% RSLogix 500 project Project_8.RSS, saved by version 8.30.00.16 %
PROJECT "UNTITLED"    % processor: Bul.1763 MicroLogix 1100 Series B %

PROGRAM FILES
  LAD 2   16 rungs

DATA FILES
  O0 OUTPUT  4 elements
  I1 INPUT  6 elements
  S2 STATUS  66 elements
  B3 BINARY  1 elements
  T4 TIMER  1 elements
  C5 COUNTER  1 elements
  R6 CONTROL  1 elements
  N7 INTEGER  7 elements
  F8 FLOAT  1 elements

LADDER 2
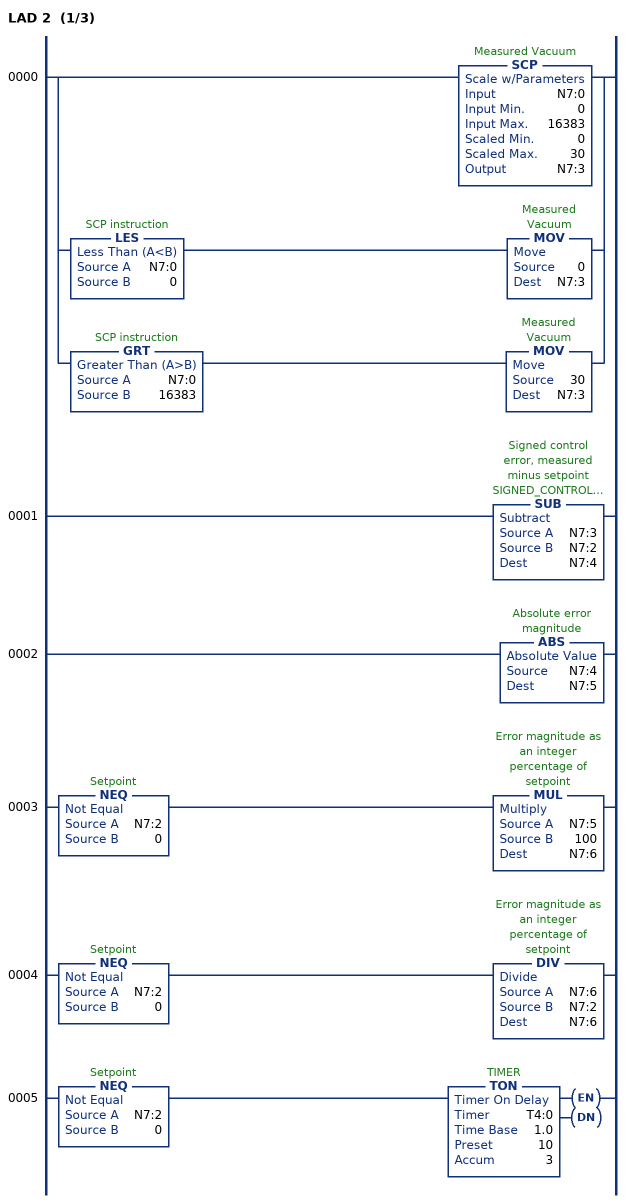
% Rung: 0 %
SOR BST SCP N7:0 0 16383 0 30 N7:3 NXB LES N7:0 0 MOV 0 N7:3 NXB GRT N7:0 16383 MOV 30 N7:3 BND EOR
%   N7:0  "SCP instruction" %
%   N7:3  "Measured Vacuum" %
% Rung: 1 %
SOR SUB N7:3 N7:2 N7:4 EOR
%   N7:3  "Measured Vacuum" %
%   N7:2  "Setpoint" %
%   N7:4  SIGNED_CONTROL_ERROR  "Signed control error, measured minus setpoint" %
% Rung: 2 %
SOR ABS N7:4 N7:5 EOR
%   N7:4  SIGNED_CONTROL_ERROR  "Signed control error, measured minus setpoint" %
%   N7:5  "Absolute error magnitude" %
% Rung: 3 %
SOR NEQ N7:2 0 MUL N7:5 100 N7:6 EOR
%   N7:2  "Setpoint" %
%   N7:5  "Absolute error magnitude" %
%   N7:6  "Error magnitude as an integer percentage of setpoint" %
% Rung: 4 %
SOR NEQ N7:2 0 DIV N7:6 N7:2 N7:6 EOR
%   N7:2  "Setpoint" %
%   N7:6  "Error magnitude as an integer percentage of setpoint" %
% Rung: 5 %
SOR NEQ N7:2 0 TON T4:0 1.0 10 3 EOR
%   N7:2  "Setpoint" %
%   T4:0  TIMER %

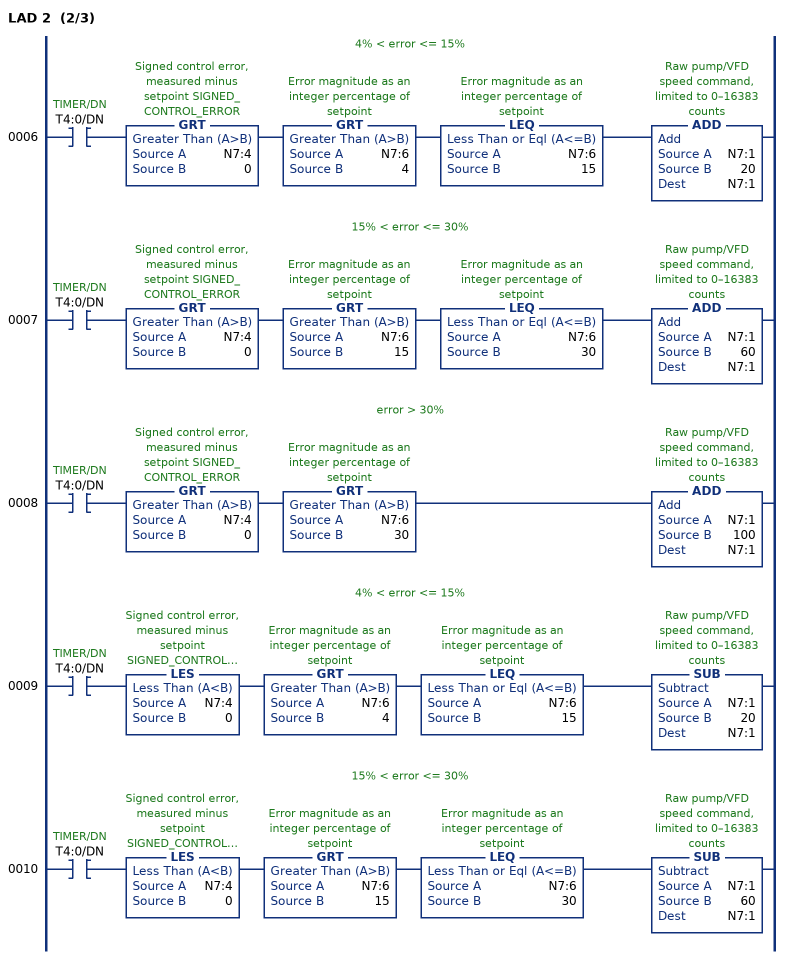
% Rung: 6 %
% 4% < error <= 15% %
SOR XIC T4:0/DN GRT N7:4 0 GRT N7:6 4 LEQ N7:6 15 ADD N7:1 20 N7:1 EOR
%   T4:0  TIMER %
%   N7:4  SIGNED_CONTROL_ERROR  "Signed control error, measured minus setpoint" %
%   N7:6  "Error magnitude as an integer percentage of setpoint" %
%   N7:1  "Raw pump/VFD speed command, limited to 0–16383 counts" %
% Rung: 7 %
% 15% < error <= 30% %
SOR XIC T4:0/DN GRT N7:4 0 GRT N7:6 15 LEQ N7:6 30 ADD N7:1 60 N7:1 EOR
%   T4:0  TIMER %
%   N7:4  SIGNED_CONTROL_ERROR  "Signed control error, measured minus setpoint" %
%   N7:6  "Error magnitude as an integer percentage of setpoint" %
%   N7:1  "Raw pump/VFD speed command, limited to 0–16383 counts" %
% Rung: 8 %
% error > 30% %
SOR XIC T4:0/DN GRT N7:4 0 GRT N7:6 30 ADD N7:1 100 N7:1 EOR
%   T4:0  TIMER %
%   N7:4  SIGNED_CONTROL_ERROR  "Signed control error, measured minus setpoint" %
%   N7:6  "Error magnitude as an integer percentage of setpoint" %
%   N7:1  "Raw pump/VFD speed command, limited to 0–16383 counts" %
% Rung: 9 %
% 4% < error <= 15% %
SOR XIC T4:0/DN LES N7:4 0 GRT N7:6 4 LEQ N7:6 15 SUB N7:1 20 N7:1 EOR
%   T4:0  TIMER %
%   N7:4  SIGNED_CONTROL_ERROR  "Signed control error, measured minus setpoint" %
%   N7:6  "Error magnitude as an integer percentage of setpoint" %
%   N7:1  "Raw pump/VFD speed command, limited to 0–16383 counts" %
% Rung: 10 %
% 15% < error <= 30% %
SOR XIC T4:0/DN LES N7:4 0 GRT N7:6 15 LEQ N7:6 30 SUB N7:1 60 N7:1 EOR
%   T4:0  TIMER %
%   N7:4  SIGNED_CONTROL_ERROR  "Signed control error, measured minus setpoint" %
%   N7:6  "Error magnitude as an integer percentage of setpoint" %
%   N7:1  "Raw pump/VFD speed command, limited to 0–16383 counts" %

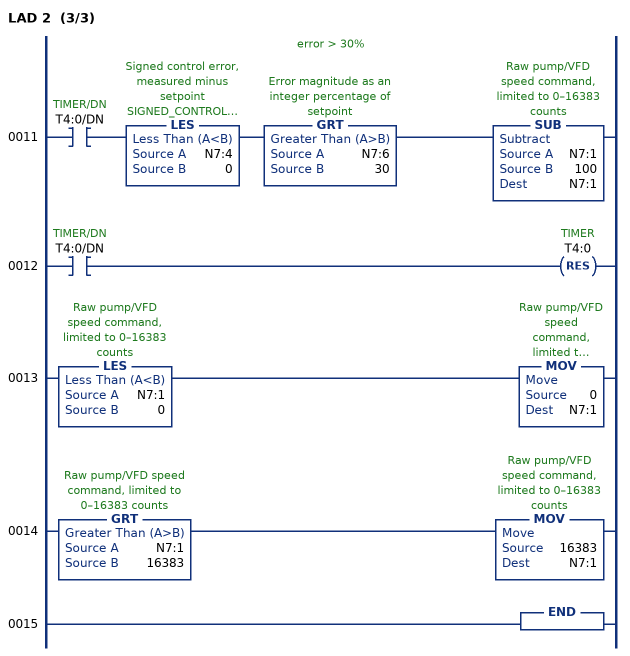
% Rung: 11 %
% error > 30% %
SOR XIC T4:0/DN LES N7:4 0 GRT N7:6 30 SUB N7:1 100 N7:1 EOR
%   T4:0  TIMER %
%   N7:4  SIGNED_CONTROL_ERROR  "Signed control error, measured minus setpoint" %
%   N7:6  "Error magnitude as an integer percentage of setpoint" %
%   N7:1  "Raw pump/VFD speed command, limited to 0–16383 counts" %
% Rung: 12 %
SOR XIC T4:0/DN RES T4:0 EOR
%   T4:0  TIMER %
% Rung: 13 %
SOR LES N7:1 0 MOV 0 N7:1 EOR
%   N7:1  "Raw pump/VFD speed command, limited to 0–16383 counts" %
% Rung: 14 %
SOR GRT N7:1 16383 MOV 16383 N7:1 EOR
%   N7:1  "Raw pump/VFD speed command, limited to 0–16383 counts" %
% Rung: 15 %
SOR END EOR

DATA TABLE (non-zero values as saved)
DATA T4
% .PRE .ACC %
% T4:0 % 10 3
DATA N7
% N7:0 % 4000 0 15 7 -8 8 53
